// TIA Portal V19 export
FUNCTION "FC_FW_Auftrag_Suche" : Void   // FC180, LAD
{ S7_Optimized_Access := 'TRUE' }
// stored: AutoNumber false, SetENOAutomatically false
   VAR_INPUT
      Pos1 : Int;
      Pos2 : Int;
   END_VAR
   VAR_IN_OUT
      Positionen : Array[1..30] of "UDT_Auftrag_Pos";
      Quelle : Int;
      Oldest : Real;
   END_VAR
   VAR_TEMP
      Pos : Int;
   END_VAR
BEGIN

REGION Network 1 (SCL)
   FOR #Pos := #Pos1 TO #Pos2 DO
       IF #Positionen[#Pos].Abholbar AND NOT #Positionen[#Pos].CheckSperre THEN
           IF (#Quelle = 0) OR (#Positionen[#Pos].Oldest > #Oldest) THEN
               #Quelle := #Pos;
               #Oldest := #Positionen[#Pos].Oldest;
           END_IF;
       END_IF;
   END_FOR;
END_REGION
END_FUNCTION
